PROGRAM AdsTcp_WinCE
VAR_OUTPUT
	bBusy : BOOL;
	err : BOOL;
	errid : UDINT;
END_VAR
VAR_OUTPUT
	areaSockets : ARRAY[1..6] OF POINTER TO AdsSocket; //only used for finding a socket by name, POINTER because array of REFERENCE does not exist
	
	//unlikely that each area will need communication with all other areas
	//only area 3 needs access to all areas, other areas only need access to area 3
	//AREA_1 : AdsSocket := (PrgName := 'AREA_1', AmsNetId := '1.0.131.216.1.1', AmsPort := 851);
	AREA_2 : AdsSocket := (PrgName := 'AREA_2', AmsNetId := ''(*'2.0.131.216.1.1'*), AmsPort := 851);
	//AREA_3 : AdsSocket := (PrgName := 'AREA_3', AmsNetId := '3.0.131.216.1.1', AmsPort := 851);
	//AREA_4 : AdsSocket := (PrgName := 'AREA_4', AmsNetId := '4.0.131.216.1.1', AmsPort := 851);
	//AREA_5 : AdsSocket := (PrgName := 'AREA_5', AmsNetId := '5.0.131.216.1.1', AmsPort := 851);
	//AREA_6 : AdsSocket := (PrgName := 'AREA_6', AmsNetId := '6.0.131.216.1.1', AmsPort := 851);
END_VAR
VAR	
	socket : REFERENCE TO AdsSocket;
	(*
	transmissons are queued into AdsTcpUnit, where all the preset sockets are
	to send a transmission, place the data and a recipient name into an AdsMessage type
	when a transmission is polled from the queue:
		if the recipient does not exist, the message contents are discarded
		if the recipient exists and is not busy writing, then the message contents are given to the socket to be written
		if the recipient is busy, then the messsage is pushed back into the queue
	*)
	
	i : INT(1..numSockets);
END_VAR
VAR CONSTANT
	numSockets : INT := 6-1;
END_VAR
(*
due to the inflexible stack size of Windows CE controllers,
this version of AdsTcp communication does not dynamically generate ADS messages into a queue to be polled cyclically
instead, modules must wait for the requested socket to finish sending its previous data before sending the next
*)

//areaSockets[1] := ADR(AREA_1);
areaSockets[2] := ADR(AREA_2);
//areaSockets[3] := ADR(AREA_3);
//areaSockets[4] := ADR(AREA_4);
//areaSockets[5] := ADR(AREA_5);
//areaSockets[6] := ADR(AREA_6);

blocks();

METHOD PRIVATE blocks : BOOL
VAR_INPUT
END_VAR
(*
AREA_1(
	PrgName=> , 
	AmsNetId=> , 
	AmsPort=> , 
	receivingData=> , 
	sendingData=> , 
	readBusy=> , 
	readError=> , 
	readErrorId=> , 
	writeBusy=> , 
	writeError=> , 
	writeErrorId=> );
*)
AREA_2(
	PrgName=> , 
	AmsNetId=> , 
	AmsPort=> , 
	receivingData=> , 
	sendingData=> , 
	readBusy=> , 
	readError=> , 
	readErrorId=> , 
	writeBusy=> , 
	writeError=> , 
	writeErrorId=> );
(*
AREA_3(
	PrgName=> , 
	AmsNetId=> , 
	AmsPort=> , 
	receivingData=> , 
	sendingData=> , 
	readBusy=> , 
	readError=> , 
	readErrorId=> , 
	writeBusy=> , 
	writeError=> , 
	writeErrorId=> );
	
AREA_4(
	PrgName=> , 
	AmsNetId=> , 
	AmsPort=> , 
	receivingData=> , 
	sendingData=> , 
	readBusy=> , 
	readError=> , 
	readErrorId=> , 
	writeBusy=> , 
	writeError=> , 
	writeErrorId=> );
	
AREA_5(
	PrgName=> , 
	AmsNetId=> , 
	AmsPort=> , 
	receivingData=> , 
	sendingData=> , 
	readBusy=> , 
	readError=> , 
	readErrorId=> , 
	writeBusy=> , 
	writeError=> , 
	writeErrorId=> );
	
AREA_6(
	PrgName=> , 
	AmsNetId=> , 
	AmsPort=> , 
	receivingData=> , 
	sendingData=> , 
	readBusy=> , 
	readError=> , 
	readErrorId=> , 
	writeBusy=> , 
	writeError=> , 
	writeErrorId=> );
*)
END_METHOD

METHOD PRIVATE findSocket : REFERENCE TO AdsSocket
VAR_INPUT
	recipient : STRING;
END_VAR
FOR i:=1 TO numSockets BY 1 DO
	IF areaSockets[i] <> 0 AND_THEN areaSockets[i]^.PrgName = recipient THEN //socket is valid, and socket name matches recipient
		findSocket REF= areaSockets[i]^;
		RETURN;
	END_IF
END_FOR
END_METHOD

METHOD pollData : BOOL
VAR_INPUT
	//remotePrgName : STRING;
	buffer : PVOID;
	bufferSize : UDINT;
	
	data : PVOID;
	dataSize : UDINT;
END_VAR
MEMCPY(buffer, data, MIN(dataSize, bufferSize));
MEMSET(data, 0, dataSize);
END_METHOD

METHOD retrieveData : BOOL
VAR_INPUT
	name : STRING;
END_VAR
VAR_IN_OUT
	genericBuffer : ARRAY[*] OF BYTE;
END_VAR
VAR
	bufferSize : DINT;
	
	//reqHandle : REFERENCE TO AdsHandle;
END_VAR
(*
bufferSize := UPPER_BOUND(genericBuffer, 1) - LOWER_BOUND(genericBuffer, 1) + 1;

reqHandle REF= findHandle('CLIENT_1');

IF __ISVALIDREF(reqHandle) THEN
	genericBuffer := ADR(reqHandle.genericBuffer);
	stDemo := reqHandle.receiverStDemo;
END_IF
*)
END_METHOD

METHOD sendMessage : BOOL
VAR_INPUT
	recipient : STRING;
	data : REFERENCE TO AdsData;
END_VAR
VAR
	//socket : REFERENCE TO AdsSocket;
END_VAR
socket REF= findSocket(recipient := recipient);

IF __ISVALIDREF(socket) AND_THEN NOT socket.writeBusy THEN
	socket.send(data := data);
	sendMessage := TRUE;
END_IF
END_METHOD

END_PROGRAM

(* stored: Version 1.1.0.1, ProductVersion 3.1.4024.11
   POU AdsTcp_WinCE: Id {fdbfe87f-1184-47dd-b08b-0750e1c8692f}, SpecialFunc None
   Method blocks: Id {84a4da9e-7305-47f8-b050-02c3484c700e}
   Method findSocket: Id {d8b3993d-426a-4e5d-a36f-587468829b99}
   Method pollData: Id {6144f990-d98d-4185-80a9-4af55f74b676}
   Method retrieveData: Id {2cc70b80-d3aa-4967-83df-e2063544db71}
   Method sendMessage: Id {b6eb2d2a-cefe-4778-a48c-87e2bc9a1963} *)
